FUNCTION ModelInfoEquals : BOOL
VAR_INPUT
    a : DUT_ModelInfo;
    b : DUT_ModelInfo;
END_VAR
VAR
    i : INT;
END_VAR


ModelInfoEquals := TRUE;
IF a.sName <> b.sName THEN
    ModelInfoEquals := FALSE;
END_IF
FOR i := 0 TO cMaxTypeNo - 1 DO
    IF a.abType[i] <> b.abType[i] THEN
        ModelInfoEquals := FALSE;
    END_IF
    IF a.aiType[i] <> b.aiType[i] THEN
        ModelInfoEquals := FALSE;
    END_IF
END_FOR
FOR i := 0 TO cMaxAxisNo - 1 DO
    IF a.arPosition[i] <> b.arPosition[i] THEN
        ModelInfoEquals := FALSE;
    END_IF
    IF a.arSpeed[i] <> b.arSpeed[i] THEN
        ModelInfoEquals := FALSE;
    END_IF
END_FOR

END_FUNCTION

(* stored: Version 1.1.0.1
   POU ModelInfoEquals: Id {e2fc5e56-b115-4c13-b67c-cce89fbdd5a3}, SpecialFunc None *)
